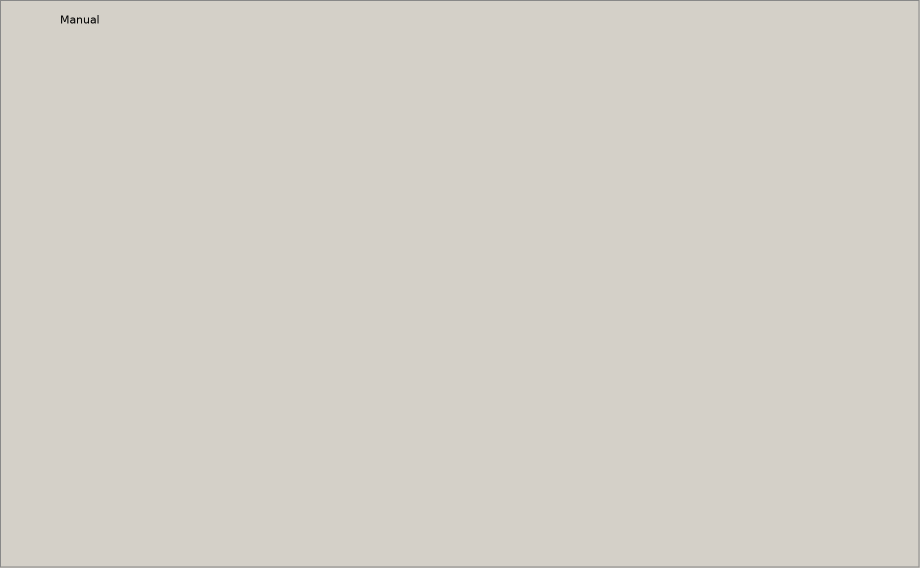
VISUALIZATION Manual  // 920x568
    Label (5,5 150x30), "Manual"
END_VISUALIZATION

(* stored: Version 1.1.0.1
   Visu Manual: Id {9b0395f1-73c7-4e6f-9dea-9dcd7208ab8b} *)
